(* Visualisation MANUAL_ST00_2
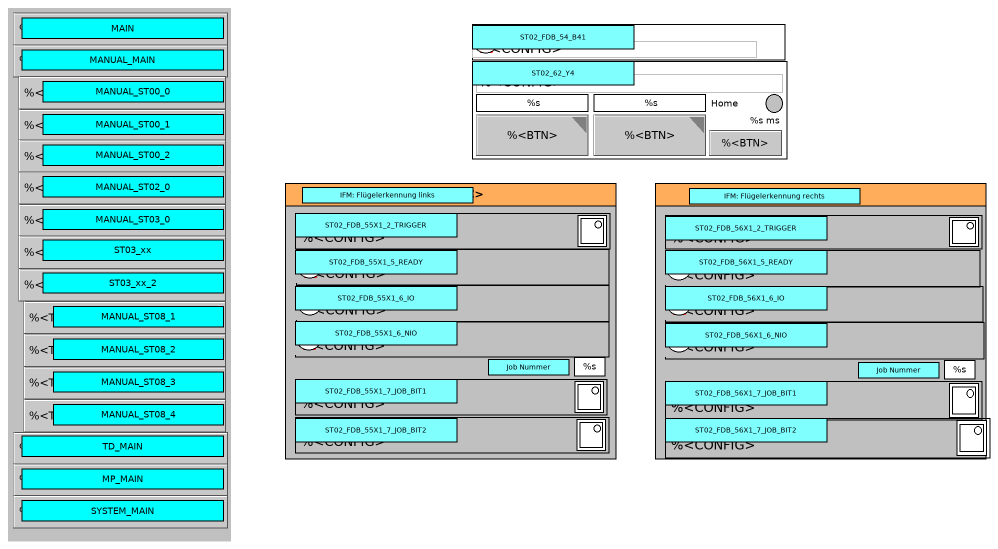
rectangle at (280,290)-(611,313): text "%<BASIC>"; shows 'IFM_Flügelerkennung_links'
rectangle at (650,290)-(981,313): text "%<BASIC>"; shows 'IFM_Flügelerkennung_rechts'
embedded screen at (3,115)-(226,648): M0000_Manual
embedded screen at (291,356)-(604,392): VDIGIN
embedded screen at (291,392)-(604,429): VDIGIN
embedded screen at (290,428)-(604,464): VDIGIN
embedded screen at (660,322)-(977,356): VDIGOUT_SMAL
embedded screen at (660,357)-(975,394): VDIGIN
embedded screen at (660,393)-(978,429): VDIGIN
embedded screen at (660,429)-(979,466): VDIGIN
embedded screen at (467,131)-(780,167): VDIGIN
embedded screen at (467,168)-(782,266): ZLIB_VALVE_1_SENSORS
embedded screen at (290,320)-(605,356): VDIGOUT_SMAL
embedded screen at (290,486)-(602,522): VDIGOUT_SMAL
embedded screen at (290,524)-(604,560): VDIGOUT_SMAL
embedded screen at (660,488)-(977,527): VDIGOUT_SMAL
embedded screen at (660,525)-(985,565): VDIGOUT_SMAL
rectangle at (297,294)-(468,310): text "IFM: Flügelerkennung links"; invisible if TRUE
rectangle at (684,295)-(855,311): text "IFM: Flügelerkennung rechts"; invisible if TRUE
rectangle at (481,464)-(562,483): text "%<BASIC>"; shows 'Job Nummer'
rectangle at (569,464)-(600,483): text "%s"; shows TD.IFM_CamProgNo; editable 0..3
rectangle at (483,466)-(564,482): text "Job Nummer"; invisible if TRUE
rectangle at (851,467)-(932,486): text "%<BASIC>"; shows 'Job Nummer'
rectangle at (939,467)-(970,486): text "%s"; shows TD.IFM_CamProgNo; editable 0..3
rectangle at (853,469)-(934,485): text "Job Nummer"; invisible if TRUE
rectangle at (290,486)-(452,510): text "ST02_FDB_55X1_7_JOB_BIT1"; invisible if TRUE
rectangle at (290,525)-(452,549): text "ST02_FDB_55X1_7_JOB_BIT2"; invisible if TRUE
rectangle at (290,428)-(452,452): text "ST02_FDB_55X1_6_NIO"; invisible if TRUE
rectangle at (290,393)-(452,417): text "ST02_FDB_55X1_6_IO"; invisible if TRUE
rectangle at (290,357)-(452,381): text "ST02_FDB_55X1_5_READY"; invisible if TRUE
rectangle at (290,320)-(452,344): text "ST02_FDB_55X1_2_TRIGGER"; invisible if TRUE
rectangle at (660,488)-(822,512): text "ST02_FDB_56X1_7_JOB_BIT1"; invisible if TRUE
rectangle at (660,525)-(822,549): text "ST02_FDB_56X1_7_JOB_BIT2"; invisible if TRUE
rectangle at (660,430)-(822,454): text "ST02_FDB_56X1_6_NIO"; invisible if TRUE
rectangle at (660,393)-(822,417): text "ST02_FDB_56X1_6_IO"; invisible if TRUE
rectangle at (660,357)-(822,381): text "ST02_FDB_56X1_5_READY"; invisible if TRUE
rectangle at (660,323)-(822,347): text "ST02_FDB_56X1_2_TRIGGER"; invisible if TRUE
rectangle at (467,132)-(629,156): text "ST02_FDB_54_B41"; invisible if TRUE
rectangle at (467,168)-(629,192): text "ST02_62_Y4"; invisible if TRUE
2 more shapes without text or variables
*)

(* Visualisation MANUAL_ST02_0
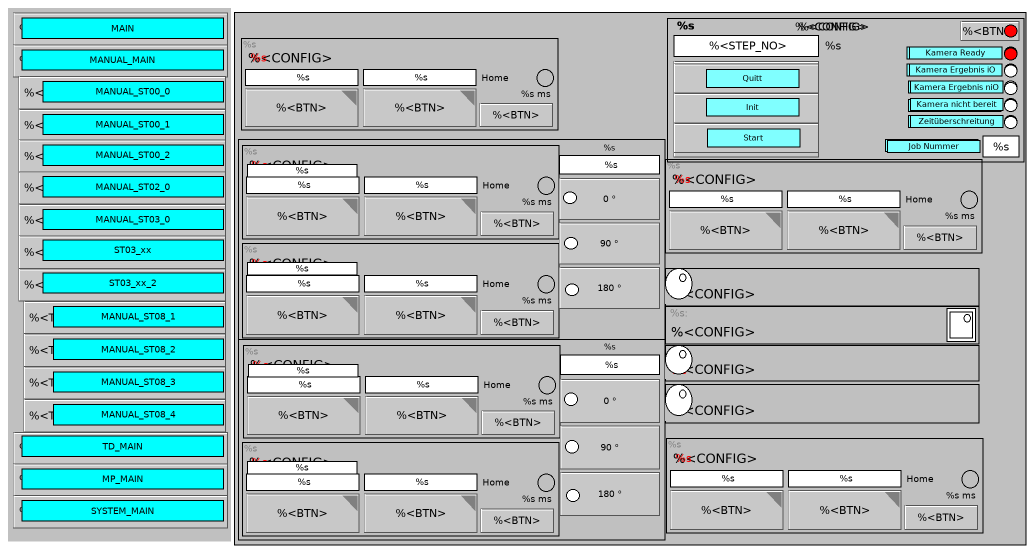
embedded screen at (3,115)-(226,648): M0000_Manual
rectangle at (233,246)-(660,447): alarm colour if ST02_62_Y6.SensorWorkIn[1].SensorSignal
rectangle at (233,446)-(660,647): alarm colour if ST02_62_Y6.SensorInitIn[1].SensorSignal
embedded screen at (660,413)-(974,451): VDIGOUT_SMAL
embedded screen at (236,145)-(553,237): ZLIB_VALVE_1_SENSORS
embedded screen at (660,452)-(974,488): VDIGIN
embedded screen at (237,350)-(554,445): ZLIB_VALVE_1_SENSORS
embedded screen at (237,252)-(554,346): ZLIB_VALVE_1_SENSORS
embedded screen at (237,549)-(554,643): ZLIB_VALVE_1_SENSORS
embedded screen at (238,452)-(555,545): ZLIB_VALVE_1_SENSORS
embedded screen at (552,249)-(657,422): ZLIB_Schwenkarm
embedded screen at (553,448)-(657,629): ZLIB_Schwenkarm
rectangle at (242,568)-(352,581): text "%s"; shows 'ST02_DT_61_B51'; alarm colour if ST02_DT_61_B51.ValveSensor
rectangle at (243,471)-(353,484): text "%s"; shows 'ST02_DT_61_B51'; alarm colour if ST02_DT_61_B51.ValveSensor
rectangle at (242,369)-(352,382): text "%s"; shows 'ST02_DT_61_B21'; alarm colour if ST02_DT_61_B21.ValveSensor
rectangle at (242,271)-(352,284): text "%s"; shows 'ST02_DT_61_B21'; alarm colour if ST02_DT_61_B21.ValveSensor
embedded screen at (660,375)-(974,413): VDIGIN
embedded screen at (660,491)-(974,530): VDIGIN
embedded screen at (661,545)-(978,640): ZLIB_VALVE_1_SENSORS
embedded screen at (660,266)-(977,360): ZLIB_VALVE_1_SENSORS
embedded screen at (662,125)-(1019,269): ZLIB_SENSOPART; invisible if MP.ST02.SensopartEthernet
embedded screen at (662,125)-(1019,269): ZLIB_SENSOPART_4; invisible if NOT MP.ST02.SensopartEthernet
1 more shapes without text or variables
*)

(* Visualisation MANUAL_ST03_0
embedded screen at (3,115)-(226,656): M0000_Manual
embedded screen at (234,123)-(549,159): VDIGIN
embedded screen at (233,161)-(844,458): ZLIB_EPSON_ROBOT
button at (244,538)-(555,574): text "%<BTN>"; shows 'Schwenkeinheit Ein'; taps ST03_ManRobotSwivelUnit.ToggleBtnOn; dynamic style Color.lightgrey, ModeSelect.Mode<>MODE_MANUAL OR NOT Robot01.RemInRunning
button at (244,462)-(555,498): text "%<BTN>"; shows 'Schwenkeinheit Aus'; taps ST03_ManRobotSwivelUnit.ToggleBtnOff; dynamic style Color.lightgrey, ModeSelect.Mode<>MODE_MANUAL OR NOT Robot01.RemInRunning
embedded screen at (244,499)-(559,536): VDIGIN
embedded screen at (244,575)-(559,612): VDIGIN
embedded screen at (244,615)-(559,652): VDIGIN; invisible if TRUE
rectangle at (244,538)-(351,557): text "Schwenkeinheit Ein"; invisible if TRUE
rectangle at (244,462)-(351,481): text "Schwenkeinheit Aus"; invisible if TRUE
rectangle at (235,124)-(407,145): text "ST03_125_F1"; invisible if TRUE
rectangle at (244,499)-(416,520): text "ST03_400_B12_6"; invisible if TRUE
rectangle at (244,575)-(416,596): text "ST03_400_B12_7"; invisible if TRUE
rectangle at (244,615)-(416,636): text "St03_120_A1_A14"; invisible if TRUE
rectangle at (0,0)-(111,51): text "%<BASIC>"; shows 'Lageerkennung'
rounded rectangle at (14,18)-(95,39): text "ERROR"
rounded rectangle at (14,18)-(95,39): text "Pos 35"; invisible if ST03_Init_AbholPos.RoboPos31 AND ST03_Init_AbholPos.RoboPos35
rounded rectangle at (14,18)-(95,39): text "Pos 31"; invisible if ST03_Init_AbholPos.RoboPos35; alarm colour if ST03_Init_AbholPos.RoboPos31
*)

(* Visualisation MANUAL_ST03_1
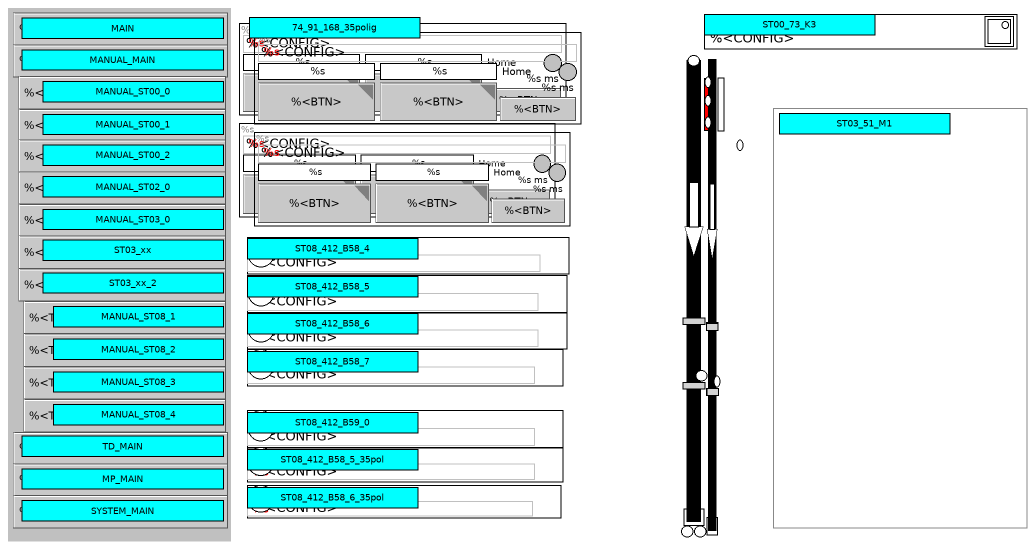
embedded screen at (3,115)-(226,648): M0000_Manual
embedded screen at (234,130)-(561,222): ZLIB_VALVE_1_SENSORS; invisible if MP.ST03.SGM_3621
embedded screen at (234,230)-(550,324): ZLIB_VALVE_1_SENSORS; invisible if MP.ST03.SGM_3621
embedded screen at (242,456)-(558,493): VDIGIN
embedded screen at (242,517)-(558,555): VDIGIN
embedded screen at (242,382)-(562,420): VDIGIN; invisible if gTypeCode = 4992
embedded screen at (242,419)-(562,456): VDIGIN; invisible if gTypeCode = 4992
embedded screen at (242,344)-(564,381): VDIGIN
embedded screen at (242,554)-(558,589): VDIGIN; invisible if gTypeCode <> 4992
embedded screen at (242,592)-(556,625): VDIGIN; invisible if gTypeCode <>4992
embedded screen at (670,162)-(711,644): ZUFUEHRUNG_35POL; invisible if gTypeCode <>4992
embedded screen at (697,166)-(738,642): ZUFUEHRUNG_74_91_168POL; invisible if gTypeCode<>360 AND gTypeCode <>379 AND gTypeCode <>489
other_LINEWIDTH at (768,215)-(1022,635): invisible if MP.ST03.SGM_3621
embedded screen at (249,139)-(576,231): ZLIB_VALVE_1_SENSORS; invisible if NOT MP.ST03.SGM_3621
embedded screen at (249,239)-(565,333): ZLIB_VALVE_1_SENSORS; invisible if NOT MP.ST03.SGM_3621
rectangle at (244,124)-(415,145): text "74_91_168_35polig"; invisible if TRUE
rectangle at (774,220)-(945,241): text "ST03_51_M1"; invisible if TRUE
rectangle at (242,345)-(413,366): text "ST08_412_B58_4"; invisible if TRUE
rectangle at (242,383)-(413,404): text "ST08_412_B58_5"; invisible if TRUE
rectangle at (242,420)-(413,441): text "ST08_412_B58_6"; invisible if TRUE
rectangle at (242,458)-(413,479): text "ST08_412_B58_7"; invisible if TRUE
rectangle at (242,519)-(413,540): text "ST08_412_B59_0"; invisible if TRUE
rectangle at (242,556)-(413,577): text "ST08_412_B58_5_35pol"; invisible if TRUE
rectangle at (242,594)-(413,615): text "ST08_412_B58_6_35pol"; invisible if TRUE
embedded screen at (699,121)-(1012,156): VDIGOUT_SMAL
rectangle at (699,121)-(870,142): text "ST00_73_K3"; invisible if TRUE
*)

(* Visualisation MANUAL_ST03_10
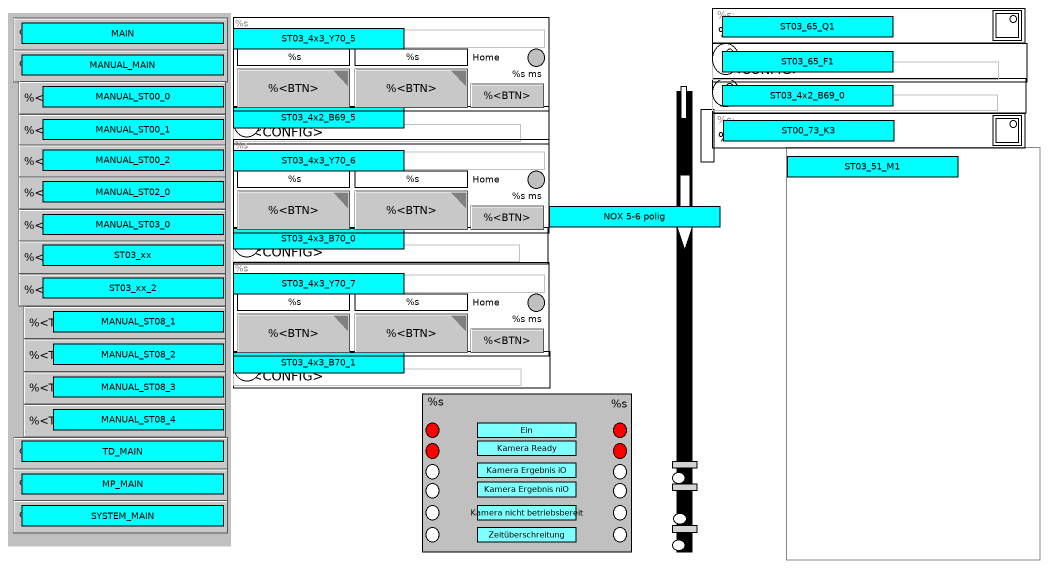
embedded screen at (3,115)-(226,648): M0000_Manual
embedded screen at (342,188)-(709,654): ZUFUEHRUNG_NOX_5_6POL; invisible if gTypeCode<>5632 AND gTypeCode<>5633
embedded screen at (228,453)-(545,490): VDIGIN
embedded screen at (707,180)-(1021,215): VDIGIN
embedded screen at (228,208)-(544,246): VDIGIN
embedded screen at (228,329)-(543,366): VDIGIN
rectangle at (544,308)-(715,329): text "NOX 5-6 polig"; invisible if TRUE
rectangle at (717,187)-(888,208): text "ST03_4x2_B69_0"; invisible if TRUE
rectangle at (228,209)-(399,230): text "ST03_4x2_B69_5"; invisible if TRUE
rectangle at (228,454)-(399,475): text "ST03_4x3_B70_1"; invisible if TRUE
rectangle at (228,330)-(399,351): text "ST03_4x3_B70_0"; invisible if TRUE
rectangle at (782,258)-(953,279): text "ST03_51_M1"; invisible if TRUE
embedded screen at (228,119)-(544,213): ZLIB_VALVE_1_SENSORS
rectangle at (228,130)-(399,151): text "ST03_4x3_Y70_5"; invisible if TRUE
embedded screen at (228,241)-(544,335): ZLIB_VALVE_1_SENSORS
rectangle at (228,252)-(399,273): text "ST03_4x3_Y70_6"; invisible if TRUE
embedded screen at (228,364)-(544,458): ZLIB_VALVE_1_SENSORS
rectangle at (228,375)-(399,396): text "ST03_4x3_Y70_7"; invisible if TRUE
embedded screen at (707,110)-(1020,145): VDIGOUT_SMAL
rectangle at (717,118)-(888,139): text "ST03_65_Q1"; invisible if TRUE
embedded screen at (707,145)-(1022,184): VDIGIN
rectangle at (717,153)-(888,174): text "ST03_65_F1"; invisible if TRUE
embedded screen at (707,215)-(1020,250): VDIGOUT_SMAL
rectangle at (718,222)-(889,243): text "ST00_73_K3"; invisible if TRUE
1 more shapes without text or variables
*)

(* Visualisation MANUAL_ST03_10_2
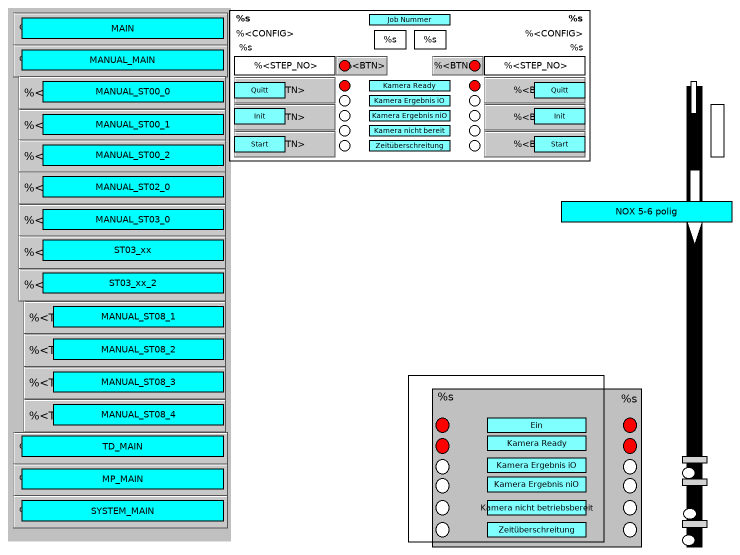
embedded screen at (3,115)-(226,648): M0000_Manual
embedded screen at (352,188)-(719,654): ZUFUEHRUNG_NOX_5_6POL; invisible if gTypeCode<>5632 AND gTypeCode<>5633
rectangle at (556,308)-(727,329): text "NOX 5-6 polig"; invisible if TRUE
embedded screen at (224,117)-(585,268): ZLIB_SENSOPART_4_2
1 more shapes without text or variables
*)

(* Visualisation MANUAL_ST03_11
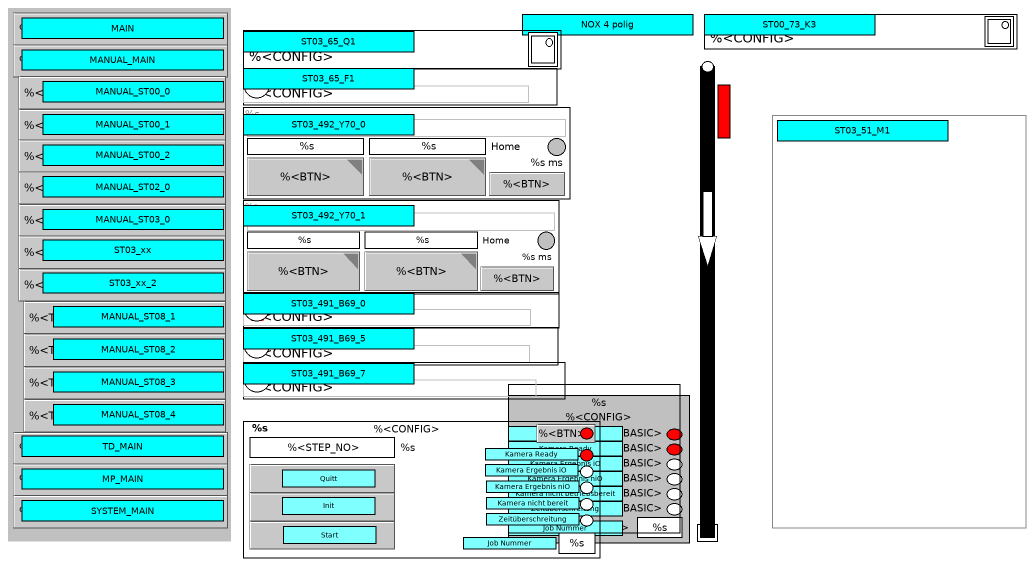
embedded screen at (3,115)-(226,648): M0000_Manual
embedded screen at (238,214)-(565,306): ZLIB_VALVE_1_SENSORS
embedded screen at (238,307)-(554,401): ZLIB_VALVE_1_SENSORS
embedded screen at (238,399)-(554,435): VDIGIN
embedded screen at (238,434)-(553,472): VDIGIN
embedded screen at (503,168)-(725,650): ZUFUEHRUNG_NOX_4POL; invisible if gTypeCode<>5631
rectangle at (517,121)-(688,142): text "NOX 4 polig"; invisible if TRUE
rectangle at (238,312)-(409,333): text "ST03_492_Y70_1"; invisible if TRUE
rectangle at (238,221)-(409,242): text "ST03_492_Y70_0"; invisible if TRUE
rectangle at (238,400)-(409,421): text "ST03_491_B69_0"; invisible if TRUE
rectangle at (238,435)-(409,456): text "ST03_491_B69_5"; invisible if TRUE
rectangle at (772,227)-(943,248): text "ST03_51_M1"; invisible if TRUE
embedded screen at (238,137)-(556,176): VDIGOUT_SMAL
rectangle at (238,138)-(409,159): text "ST03_65_Q1"; invisible if TRUE
embedded screen at (238,175)-(552,212): VDIGIN
rectangle at (238,175)-(409,196): text "ST03_65_F1"; invisible if TRUE
embedded screen at (699,121)-(1012,156): VDIGOUT_SMAL
rectangle at (699,121)-(870,142): text "ST00_73_K3"; invisible if TRUE
embedded screen at (238,528)-(595,665): ZLIB_SENSOPART_4; invisible if TRUE
embedded screen at (238,469)-(560,506): VDIGIN
rectangle at (238,470)-(409,491): text "ST03_491_B69_7"; invisible if TRUE
2 more shapes without text or variables
*)

(* Visualisation MANUAL_ST03_12
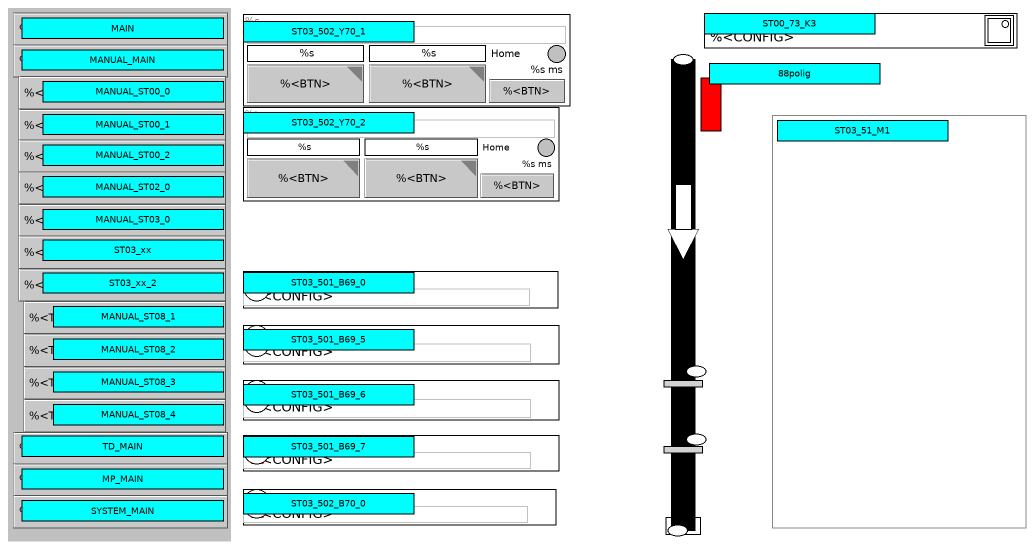
embedded screen at (3,115)-(226,648): M0000_Manual
embedded screen at (238,121)-(565,213): ZLIB_VALVE_1_SENSORS
embedded screen at (238,214)-(554,308): ZLIB_VALVE_1_SENSORS
embedded screen at (238,542)-(554,578): VDIGIN
embedded screen at (238,596)-(551,632): VDIGIN
embedded screen at (646,161)-(716,643): ZUFUEHRUNG_88POL; invisible if gTypeCode<>5731
rectangle at (704,170)-(875,191): text "88polig"; invisible if TRUE
rectangle at (238,219)-(409,240): text "ST03_502_Y70_2"; invisible if TRUE
rectangle at (238,128)-(409,149): text "ST03_502_Y70_1"; invisible if TRUE
rectangle at (238,543)-(409,564): text "ST03_501_B69_7"; invisible if TRUE
rectangle at (238,600)-(409,621): text "ST03_502_B70_0"; invisible if TRUE
rectangle at (772,227)-(943,248): text "ST03_51_M1"; invisible if TRUE
embedded screen at (238,487)-(554,527): VDIGIN
embedded screen at (238,378)-(553,415): VDIGIN
embedded screen at (238,432)-(554,471): VDIGIN
rectangle at (238,379)-(409,400): text "ST03_501_B69_0"; invisible if TRUE
rectangle at (238,436)-(409,457): text "ST03_501_B69_5"; invisible if TRUE
rectangle at (238,491)-(409,512): text "ST03_501_B69_6"; invisible if TRUE
embedded screen at (699,120)-(1012,155): VDIGOUT_SMAL
rectangle at (699,120)-(870,141): text "ST00_73_K3"; invisible if TRUE
1 more shapes without text or variables
*)

(* Visualisation MANUAL_ST03_13
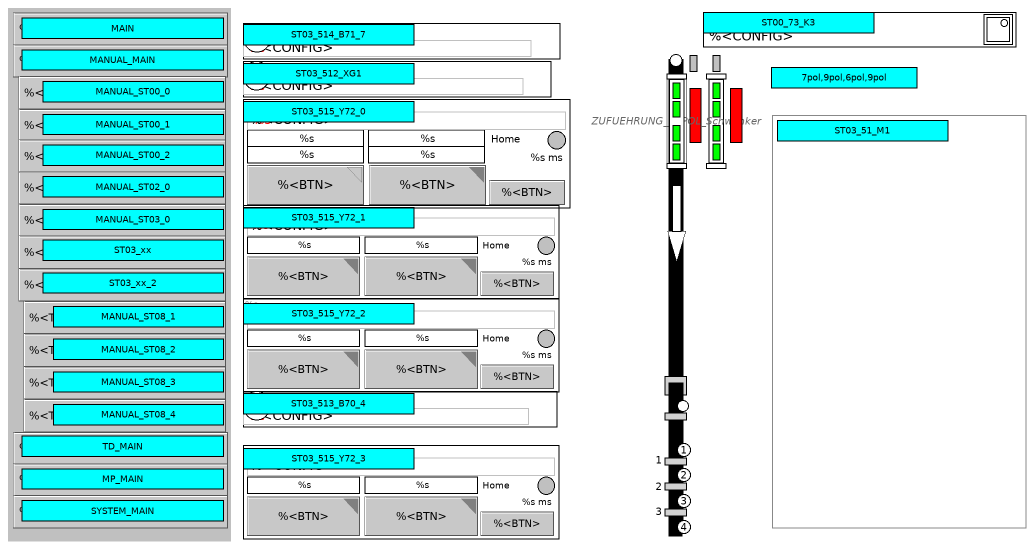
embedded screen at (3,115)-(226,648): M0000_Manual
embedded screen at (238,312)-(554,406): ZLIB_VALVE_1_SENSORS
embedded screen at (238,130)-(555,166): VDIGIN
embedded screen at (646,161)-(737,643): ZUFUEHRUNG_7POL; invisible if gTypeCode<>575  AND gTypeCode<>5753  AND gTypeCode<>5754  AND gTypeCode<>5755
rectangle at (766,174)-(912,195): text "7pol,9pol,6pol,9pol"; invisible if TRUE
rectangle at (238,314)-(409,335): text "ST03_515_Y72_1"; invisible if TRUE
rectangle at (238,131)-(409,152): text "ST03_514_B71_7"; invisible if TRUE
rectangle at (772,227)-(943,248): text "ST03_51_M1"; invisible if TRUE
embedded screen at (238,168)-(546,204): VDIGIN
rectangle at (238,170)-(409,191): text "ST03_512_XG1"; invisible if TRUE
embedded screen at (238,405)-(554,499): ZLIB_VALVE_1_SENSORS
embedded screen at (238,498)-(552,534): VDIGIN
rectangle at (238,410)-(409,431): text "ST03_515_Y72_2"; invisible if TRUE
rectangle at (238,500)-(409,521): text "ST03_513_B70_4"; invisible if TRUE
embedded screen at (238,552)-(554,646): ZLIB_VALVE_1_SENSORS
rectangle at (238,555)-(409,576): text "ST03_515_Y72_3"; invisible if TRUE
embedded screen at (238,206)-(565,315): ZLIB_VALVE_2_SENSORS
rectangle at (238,208)-(409,229): text "ST03_515_Y72_0"; invisible if TRUE
embedded screen at (698,119)-(1011,154): VDIGOUT_SMAL
rectangle at (698,119)-(869,140): text "ST00_73_K3"; invisible if TRUE
1 more shapes without text or variables
*)

(* Visualisation MANUAL_ST03_13_2
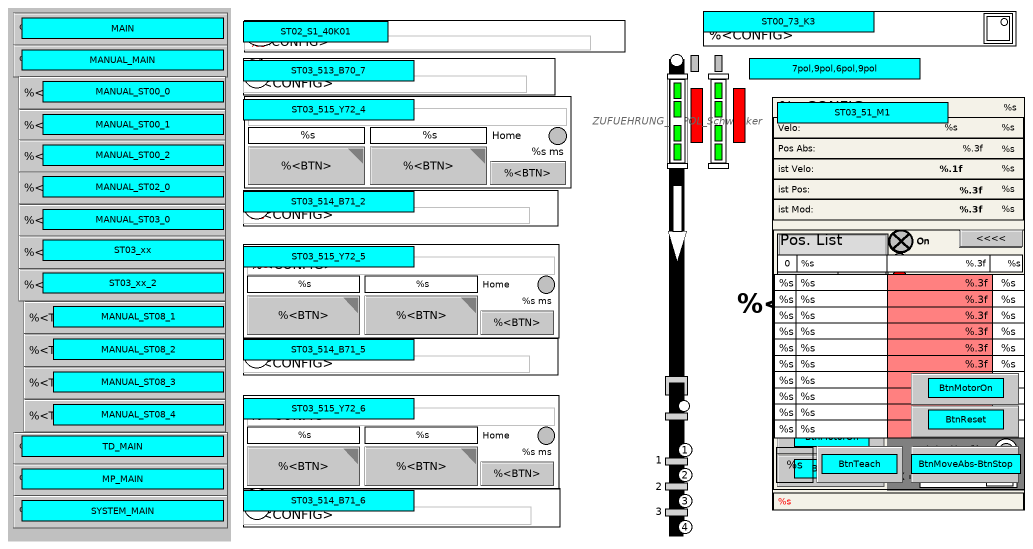
embedded screen at (3,115)-(226,648): M0000_Manual
embedded screen at (239,203)-(566,295): ZLIB_VALVE_1_SENSORS
embedded screen at (238,351)-(554,445): ZLIB_VALVE_1_SENSORS
embedded screen at (238,445)-(553,482): VDIGIN
embedded screen at (767,204)-(1021,617): ZLIB_7211_Achse
embedded screen at (646,161)-(740,643): ZUFUEHRUNG_7POL; invisible if gTypeCode<>575  AND gTypeCode<>5753  AND gTypeCode<>5754  AND gTypeCode<>5755
rectangle at (744,165)-(915,186): text "7pol,9pol,6pol,9pol"; invisible if TRUE
rectangle at (238,353)-(409,374): text "ST03_515_Y72_5"; invisible if TRUE
rectangle at (238,206)-(409,227): text "ST03_515_Y72_4"; invisible if TRUE
rectangle at (238,446)-(409,467): text "ST03_514_B71_5"; invisible if TRUE
rectangle at (772,209)-(943,230): text "ST03_51_M1"; invisible if TRUE
embedded screen at (238,165)-(550,202): VDIGIN
rectangle at (238,167)-(409,188): text "ST03_513_B70_7"; invisible if TRUE
embedded screen at (238,502)-(554,596): ZLIB_VALVE_1_SENSORS
embedded screen at (238,595)-(555,634): VDIGIN
rectangle at (238,505)-(409,526): text "ST03_515_Y72_6"; invisible if TRUE
rectangle at (238,597)-(409,618): text "ST03_514_B71_6"; invisible if TRUE
embedded screen at (238,297)-(553,333): VDIGIN
rectangle at (238,298)-(409,319): text "ST03_514_B71_2"; invisible if TRUE
embedded screen at (239,127)-(620,159): VDIGIN; invisible if gTypeCode<>4991 AND gTypeCode <>312
rectangle at (238,128)-(383,149): text "ST02_S1_40K01"; invisible if TRUE
embedded screen at (698,118)-(1011,153): VDIGOUT_SMAL
rectangle at (698,118)-(869,139): text "ST00_73_K3"; invisible if TRUE
*)

(* Visualisation MANUAL_ST03_14
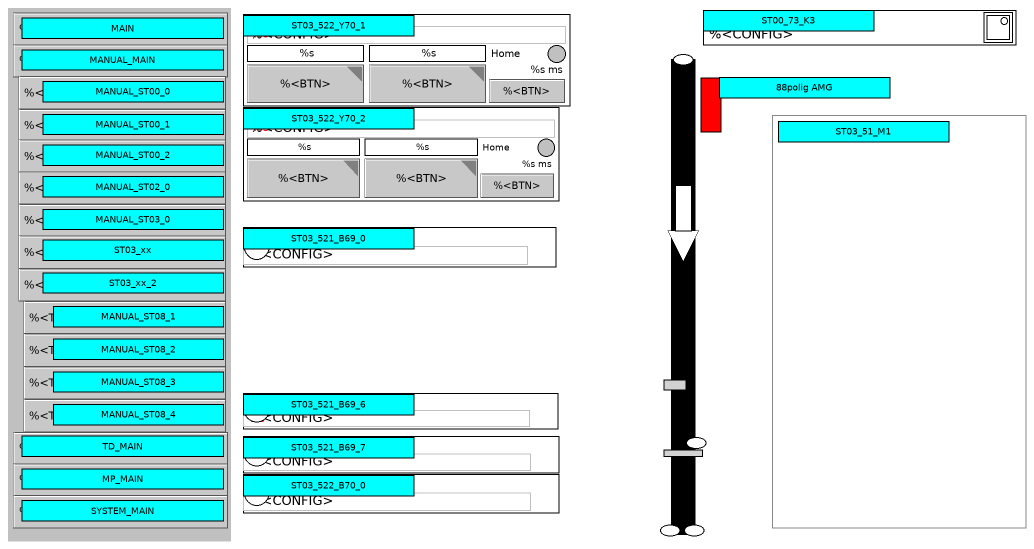
embedded screen at (3,115)-(226,648): M0000_Manual
embedded screen at (238,121)-(565,213): ZLIB_VALVE_1_SENSORS
embedded screen at (238,214)-(554,308): ZLIB_VALVE_1_SENSORS
embedded screen at (238,543)-(554,580): VDIGIN
embedded screen at (238,581)-(554,620): VDIGIN
embedded screen at (646,161)-(716,643): ZUFUEHRUNG_88POL_AMG; invisible if gTypeCode<>5732
rectangle at (714,184)-(885,205): text "88polig AMG"; invisible if TRUE
rectangle at (238,215)-(409,236): text "ST03_522_Y70_2"; invisible if TRUE
rectangle at (238,122)-(409,143): text "ST03_522_Y70_1"; invisible if TRUE
rectangle at (238,544)-(409,565): text "ST03_521_B69_7"; invisible if TRUE
rectangle at (238,582)-(409,603): text "ST03_522_B70_0"; invisible if TRUE
rectangle at (773,228)-(944,249): text "ST03_51_M1"; invisible if TRUE
embedded screen at (238,500)-(553,536): VDIGIN
embedded screen at (238,334)-(551,374): VDIGIN
rectangle at (238,335)-(409,356): text "ST03_521_B69_0"; invisible if TRUE
rectangle at (238,501)-(409,522): text "ST03_521_B69_6"; invisible if TRUE
embedded screen at (698,117)-(1011,152): VDIGOUT_SMAL
rectangle at (698,117)-(869,138): text "ST00_73_K3"; invisible if TRUE
1 more shapes without text or variables
*)

(* Visualisation MANUAL_ST03_15
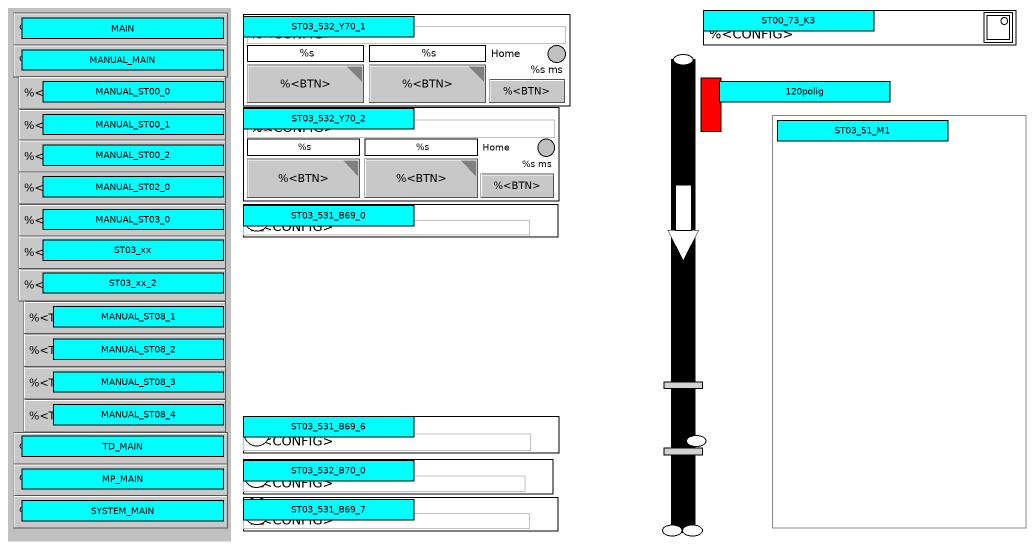
embedded screen at (3,115)-(226,648): M0000_Manual
embedded screen at (238,121)-(565,213): ZLIB_VALVE_1_SENSORS
embedded screen at (238,214)-(554,308): ZLIB_VALVE_1_SENSORS
embedded screen at (238,604)-(553,638): VDIGIN
embedded screen at (238,566)-(548,601): VDIGIN
embedded screen at (646,161)-(716,643): ZUFUEHRUNG_120POL; invisible if gTypeCode<>5771
rectangle at (714,188)-(885,209): text "120polig"; invisible if TRUE
rectangle at (238,215)-(409,236): text "ST03_532_Y70_2"; invisible if TRUE
rectangle at (238,123)-(409,144): text "ST03_532_Y70_1"; invisible if TRUE
rectangle at (238,606)-(409,627): text "ST03_531_B69_7"; invisible if TRUE
rectangle at (238,567)-(409,588): text "ST03_532_B70_0"; invisible if TRUE
rectangle at (772,227)-(943,248): text "ST03_51_M1"; invisible if TRUE
embedded screen at (238,523)-(554,560): VDIGIN
embedded screen at (238,311)-(553,344): VDIGIN
rectangle at (238,312)-(409,333): text "ST03_531_B69_0"; invisible if TRUE
rectangle at (238,523)-(409,544): text "ST03_531_B69_6"; invisible if TRUE
embedded screen at (698,117)-(1011,152): VDIGOUT_SMAL
rectangle at (698,117)-(869,138): text "ST00_73_K3"; invisible if TRUE
1 more shapes without text or variables
*)

(* Visualisation MANUAL_ST03_16
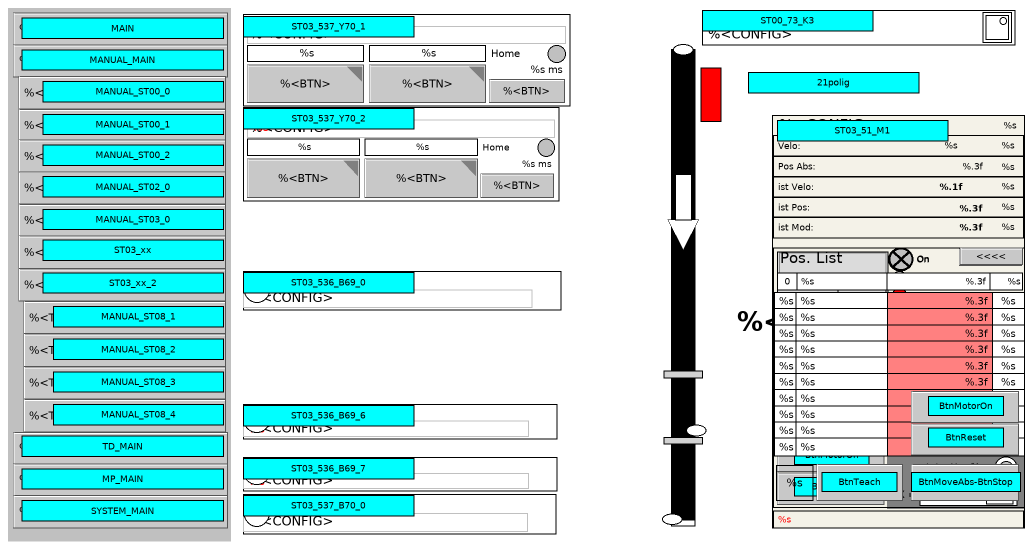
embedded screen at (3,115)-(226,648): M0000_Manual
embedded screen at (238,121)-(565,213): ZLIB_VALVE_1_SENSORS
embedded screen at (238,214)-(554,308): ZLIB_VALVE_1_SENSORS
embedded screen at (238,564)-(552,598): VDIGIN
embedded screen at (238,601)-(551,641): VDIGIN
embedded screen at (767,222)-(1021,635): ZLIB_7211_Achse
embedded screen at (646,151)-(716,633): ZUFUEHRUNG_21POL; invisible if gTypeCode<>5772
rectangle at (743,179)-(914,200): text "21polig"; invisible if TRUE
rectangle at (238,215)-(409,236): text "ST03_537_Y70_2"; invisible if TRUE
rectangle at (238,123)-(409,144): text "ST03_537_Y70_1"; invisible if TRUE
rectangle at (238,565)-(409,586): text "ST03_536_B69_7"; invisible if TRUE
rectangle at (238,602)-(409,623): text "ST03_537_B70_0"; invisible if TRUE
rectangle at (772,227)-(943,248): text "ST03_51_M1"; invisible if TRUE
embedded screen at (238,511)-(552,546): VDIGIN
embedded screen at (238,378)-(556,417): VDIGIN
rectangle at (238,379)-(409,400): text "ST03_536_B69_0"; invisible if TRUE
rectangle at (238,512)-(409,533): text "ST03_536_B69_6"; invisible if TRUE
embedded screen at (697,117)-(1010,152): VDIGOUT_SMAL
rectangle at (697,117)-(868,138): text "ST00_73_K3"; invisible if TRUE
*)

(* Visualisation MANUAL_ST03_17
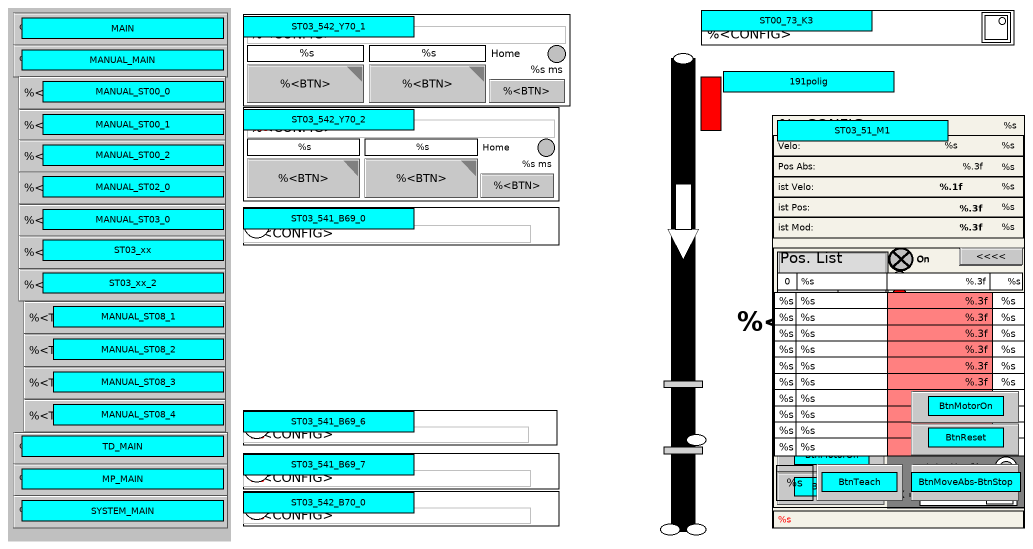
embedded screen at (3,115)-(226,648): M0000_Manual
embedded screen at (238,121)-(565,213): ZLIB_VALVE_1_SENSORS
embedded screen at (238,214)-(554,308): ZLIB_VALVE_1_SENSORS
embedded screen at (238,560)-(554,596): VDIGIN
embedded screen at (238,598)-(554,633): VDIGIN
embedded screen at (767,222)-(1021,635): ZLIB_7211_Achse
embedded screen at (646,160)-(716,642): ZUFUEHRUNG_191POL; invisible if gTypeCode<>580
rectangle at (718,178)-(889,199): text "191polig"; invisible if TRUE
rectangle at (238,216)-(409,237): text "ST03_542_Y70_2"; invisible if TRUE
rectangle at (238,123)-(409,144): text "ST03_542_Y70_1"; invisible if TRUE
rectangle at (238,561)-(409,582): text "ST03_541_B69_7"; invisible if TRUE
rectangle at (238,599)-(409,620): text "ST03_542_B70_0"; invisible if TRUE
rectangle at (772,227)-(943,248): text "ST03_51_M1"; invisible if TRUE
embedded screen at (238,517)-(552,552): VDIGIN
embedded screen at (238,314)-(554,352): VDIGIN
rectangle at (238,315)-(409,336): text "ST03_541_B69_0"; invisible if TRUE
rectangle at (238,518)-(409,539): text "ST03_541_B69_6"; invisible if TRUE
embedded screen at (696,117)-(1009,152): VDIGOUT_SMAL
rectangle at (696,117)-(867,138): text "ST00_73_K3"; invisible if TRUE
*)

(* Visualisation MANUAL_ST03_18
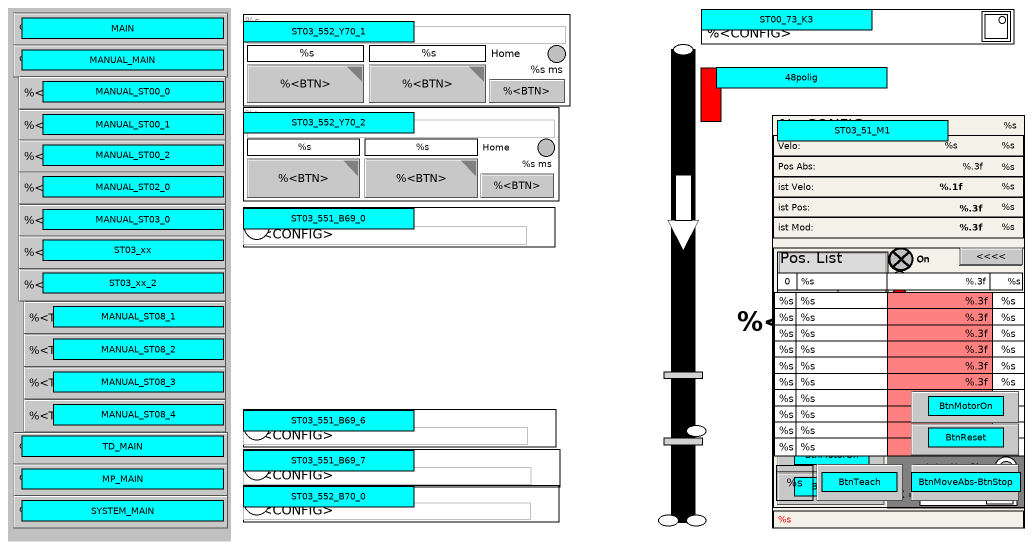
embedded screen at (3,115)-(226,648): M0000_Manual
embedded screen at (238,121)-(565,213): ZLIB_VALVE_1_SENSORS
embedded screen at (238,214)-(554,308): ZLIB_VALVE_1_SENSORS
embedded screen at (238,556)-(555,594): VDIGIN
embedded screen at (238,592)-(554,629): VDIGIN
embedded screen at (767,222)-(1021,635): ZLIB_7211_Achse
embedded screen at (646,151)-(716,633): ZUFUEHRUNG_48POL; invisible if gTypeCode<>5832
rectangle at (711,174)-(882,195): text "48polig"; invisible if TRUE
rectangle at (238,219)-(409,240): text "ST03_552_Y70_2"; invisible if TRUE
rectangle at (238,128)-(409,149): text "ST03_552_Y70_1"; invisible if TRUE
rectangle at (238,557)-(409,578): text "ST03_551_B69_7"; invisible if TRUE
rectangle at (238,593)-(409,614): text "ST03_552_B70_0"; invisible if TRUE
rectangle at (772,227)-(943,248): text "ST03_51_M1"; invisible if TRUE
embedded screen at (238,516)-(551,554): VDIGIN
embedded screen at (238,314)-(550,354): VDIGIN
rectangle at (238,315)-(409,336): text "ST03_551_B69_0"; invisible if TRUE
rectangle at (238,517)-(409,538): text "ST03_551_B69_6"; invisible if TRUE
embedded screen at (696,116)-(1009,151): VDIGOUT_SMAL
rectangle at (696,116)-(867,137): text "ST00_73_K3"; invisible if TRUE
*)

(* Visualisation MANUAL_ST03_19
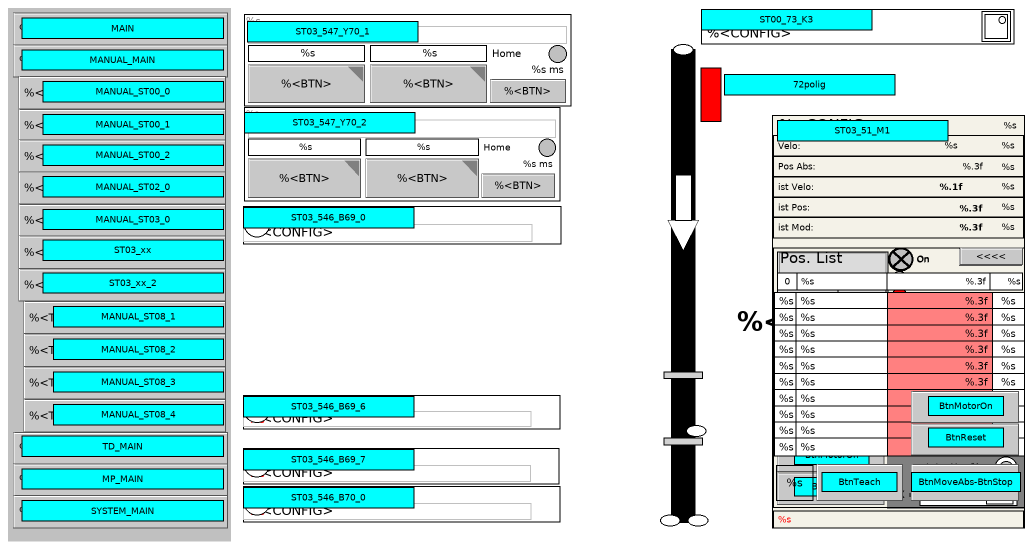
embedded screen at (3,115)-(226,648): M0000_Manual
embedded screen at (239,121)-(566,213): ZLIB_VALVE_1_SENSORS
embedded screen at (239,214)-(555,308): ZLIB_VALVE_1_SENSORS
embedded screen at (238,555)-(554,591): VDIGIN
embedded screen at (238,593)-(555,629): VDIGIN
embedded screen at (767,222)-(1021,635): ZLIB_7211_Achse
embedded screen at (646,151)-(716,633): ZUFUEHRUNG_72POL; invisible if gTypeCode<>5831
rectangle at (719,181)-(890,202): text "72polig"; invisible if TRUE
rectangle at (239,219)-(410,240): text "ST03_547_Y70_2"; invisible if TRUE
rectangle at (242,128)-(413,149): text "ST03_547_Y70_1"; invisible if TRUE
rectangle at (238,556)-(409,577): text "ST03_546_B69_7"; invisible if TRUE
rectangle at (238,594)-(409,615): text "ST03_546_B70_0"; invisible if TRUE
rectangle at (772,227)-(943,248): text "ST03_51_M1"; invisible if TRUE
embedded screen at (238,502)-(555,536): VDIGIN
embedded screen at (238,313)-(556,351): VDIGIN
rectangle at (238,314)-(409,335): text "ST03_546_B69_0"; invisible if TRUE
rectangle at (238,503)-(409,524): text "ST03_546_B69_6"; invisible if TRUE
embedded screen at (696,116)-(1009,151): VDIGOUT_SMAL
rectangle at (696,116)-(867,137): text "ST00_73_K3"; invisible if TRUE
*)

(* Visualisation MANUAL_ST03_2
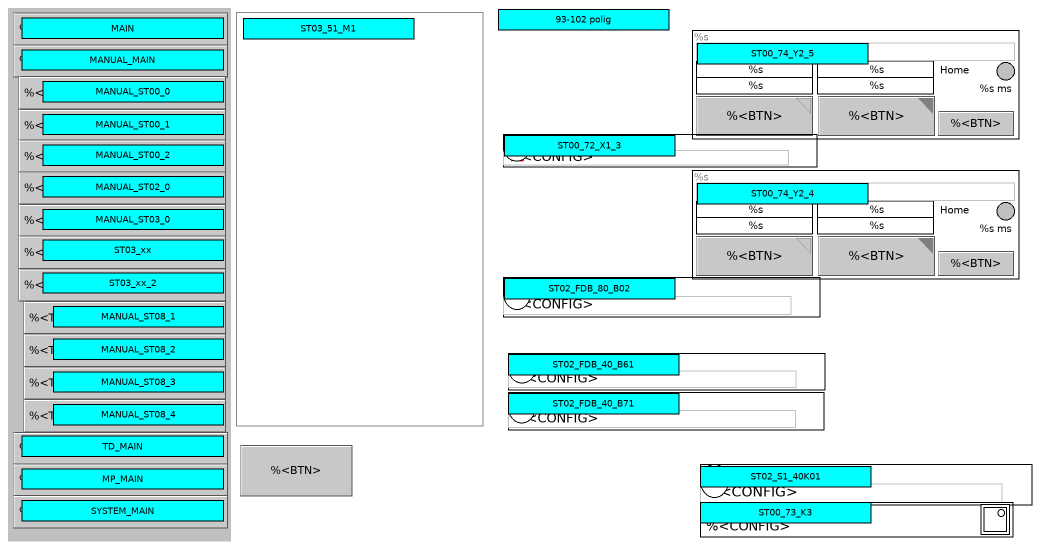
embedded screen at (3,115)-(226,648): M0000_Manual
embedded screen at (687,277)-(1014,386): ZLIB_VALVE_2_SENSORS
embedded screen at (687,137)-(1014,246): ZLIB_VALVE_2_SENSORS
other_LINEWIDTH at (231,119)-(478,533): invisible if MP.ST03.SGM_3621
embedded screen at (695,571)-(1027,612): VDIGIN
embedded screen at (498,241)-(812,274): VDIGIN
embedded screen at (498,384)-(815,424): VDIGIN
button at (235,552)-(347,603): text "%<BTN>"; shows 'TaktBand'; invisible if gTypeCode<>4991 AND gTypeCode <>312; taps ST03_Band.b_MoveRel
embedded screen at (503,460)-(820,497): VDIGIN
embedded screen at (503,499)-(819,537): VDIGIN
rectangle at (493,116)-(664,137): text "93-102 polig"; invisible if TRUE
rectangle at (238,125)-(409,146): text "ST03_51_M1"; invisible if TRUE
rectangle at (695,573)-(866,594): text "ST02_S1_40K01"; invisible if TRUE
rectangle at (503,461)-(674,482): text "ST02_FDB_40_B61"; invisible if TRUE
rectangle at (503,500)-(674,521): text "ST02_FDB_40_B71"; invisible if TRUE
rectangle at (499,385)-(670,406): text "ST02_FDB_80_B02"; invisible if TRUE
rectangle at (499,242)-(670,263): text "ST00_72_X1_3"; invisible if TRUE
rectangle at (692,150)-(863,171): text "ST00_74_Y2_5"; invisible if TRUE
rectangle at (692,290)-(863,311): text "ST00_74_Y2_4"; invisible if TRUE
embedded screen at (695,609)-(1008,644): VDIGOUT_SMAL
rectangle at (695,609)-(866,630): text "ST00_73_K3"; invisible if TRUE
*)

(* Visualisation MANUAL_ST03_20
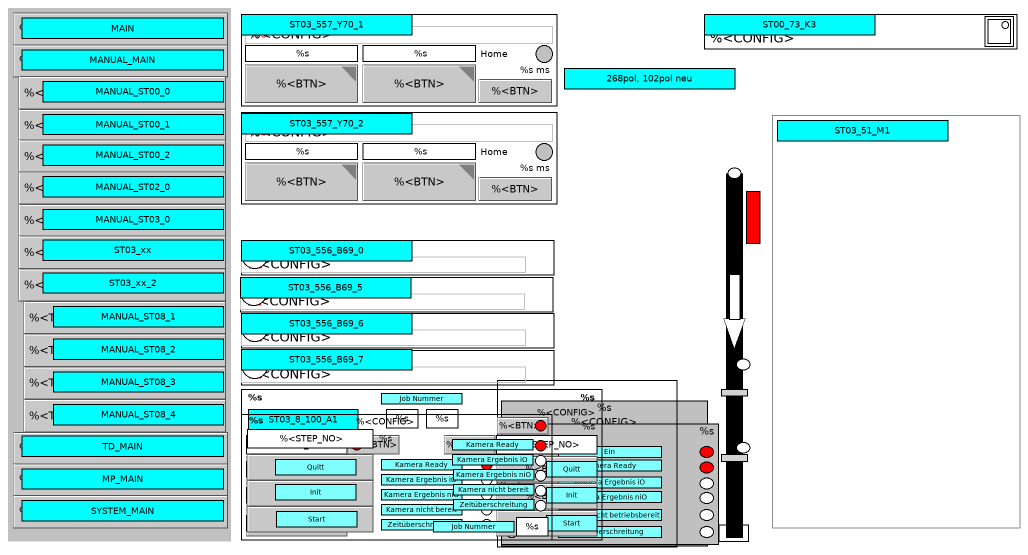
embedded screen at (3,115)-(226,648): M0000_Manual
embedded screen at (699,121)-(1012,156): VDIGOUT_SMAL
embedded screen at (236,121)-(552,213): ZLIB_VALVE_1_SENSORS
embedded screen at (236,219)-(552,311): ZLIB_VALVE_1_SENSORS
embedded screen at (496,176)-(755,653): ZUFUEHRUNG_268POL_102POL_NEU; invisible if AND gTypeCode<>4993
rectangle at (559,175)-(730,196): text "268pol, 102pol neu"; invisible if TRUE
rectangle at (236,220)-(407,241): text "ST03_557_Y70_2"; invisible if TRUE
rectangle at (236,121)-(407,142): text "ST03_557_Y70_1"; invisible if TRUE
rectangle at (699,121)-(870,142): text "ST00_73_K3"; invisible if TRUE
rectangle at (772,227)-(943,248): text "ST03_51_M1"; invisible if TRUE
embedded screen at (236,420)-(549,455): VDIGIN
embedded screen at (236,347)-(549,382): VDIGIN
rectangle at (236,347)-(407,368): text "ST03_556_B69_0"; invisible if TRUE
rectangle at (236,420)-(407,441): text "ST03_556_B69_6"; invisible if TRUE
embedded screen at (236,496)-(597,647): ZLIB_SENSOPART_4_2; invisible if gTypeCode<>4993
embedded screen at (235,384)-(548,419): VDIGIN
rectangle at (235,384)-(406,405): text "ST03_556_B69_5"; invisible if TRUE
rectangle at (243,516)-(353,537): text "ST03_8_100_A1"; invisible if TRUE
embedded screen at (236,457)-(549,492): VDIGIN
rectangle at (236,456)-(407,477): text "ST03_556_B69_7"; invisible if TRUE
embedded screen at (236,521)-(547,647): ZLIB_SENSOPART_4; invisible if gTypeCode<>5841
2 more shapes without text or variables
*)

(* Visualisation MANUAL_ST03_20_2
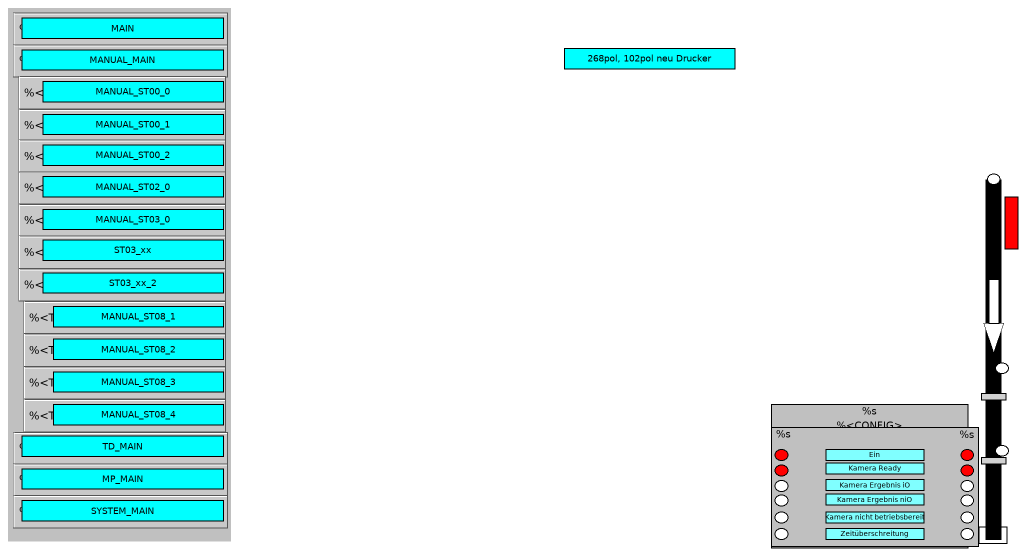
embedded screen at (766,183)-(1013,655): ZUFUEHRUNG_268POL_102POL_NEU
embedded screen at (3,115)-(226,648): M0000_Manual
rectangle at (559,155)-(730,176): text "268pol, 102pol neu Drucker"; invisible if TRUE
*)

(* Visualisation MANUAL_ST03_21
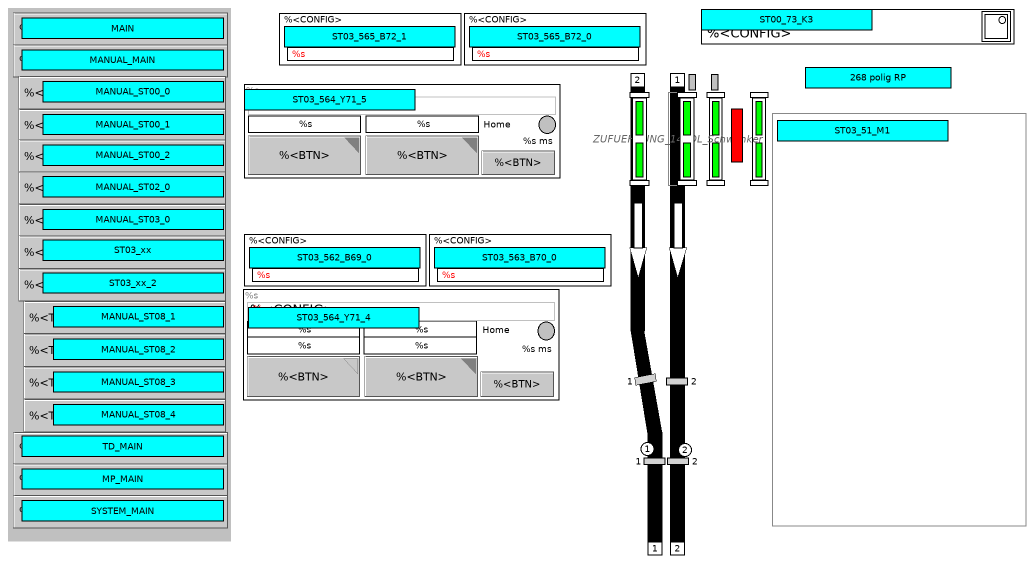
embedded screen at (3,115)-(226,648): M0000_Manual
embedded screen at (239,191)-(555,285): ZLIB_VALVE_1_SENSORS
embedded screen at (459,120)-(641,172): ZLIB_DIG_IN
embedded screen at (590,180)-(763,662): ZUFUEHRUNG_268POL_RP; invisible if gTypeCode<>5842
rectangle at (800,174)-(946,195): text "268 polig RP"; invisible if TRUE
rectangle at (239,196)-(410,217): text "ST03_564_Y71_5"; invisible if TRUE
rectangle at (464,133)-(635,154): text "ST03_565_B72_0"; invisible if TRUE
rectangle at (772,227)-(943,248): text "ST03_51_M1"; invisible if TRUE
embedded screen at (274,120)-(456,172): ZLIB_DIG_IN
rectangle at (279,133)-(450,154): text "ST03_565_B72_1"; invisible if TRUE
embedded screen at (239,341)-(421,393): ZLIB_DIG_IN
rectangle at (244,354)-(415,375): text "ST03_562_B69_0"; invisible if TRUE
embedded screen at (238,396)-(554,507): ZLIB_VALVE_2_SENSORS
rectangle at (243,414)-(414,435): text "ST03_564_Y71_4"; invisible if TRUE
embedded screen at (424,341)-(606,393): ZLIB_DIG_IN
rectangle at (429,354)-(600,375): text "ST03_563_B70_0"; invisible if TRUE
embedded screen at (696,116)-(1009,151): VDIGOUT_SMAL
rectangle at (696,116)-(867,137): text "ST00_73_K3"; invisible if TRUE
1 more shapes without text or variables
*)

(* Visualisation MANUAL_ST03_21_2
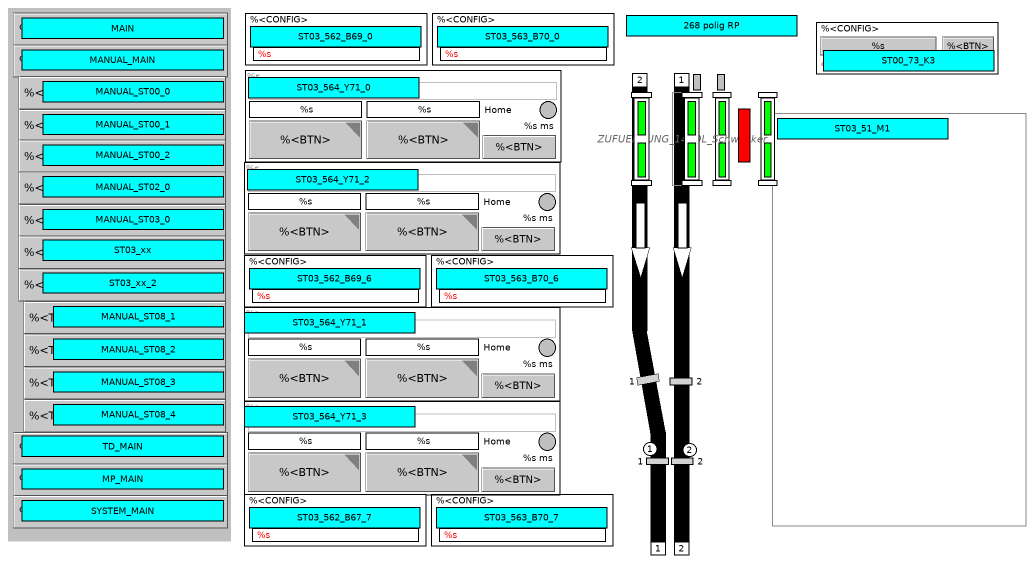
embedded screen at (3,115)-(226,648): M0000_Manual
embedded screen at (811,129)-(993,181): ZLIB_DIGOUT
embedded screen at (239,269)-(555,361): ZLIB_VALVE_1_SENSORS
embedded screen at (239,414)-(555,508): ZLIB_VALVE_1_SENSORS
embedded screen at (426,601)-(608,653): ZLIB_DIG_IN
embedded screen at (590,180)-(772,662): ZUFUEHRUNG_268POL_RP; invisible if gTypeCode<>5842
rectangle at (621,122)-(792,143): text "268 polig RP"; invisible if TRUE
rectangle at (239,419)-(410,440): text "ST03_564_Y71_1"; invisible if TRUE
rectangle at (242,276)-(413,297): text "ST03_564_Y71_2"; invisible if TRUE
rectangle at (431,614)-(602,635): text "ST03_563_B70_7"; invisible if TRUE
rectangle at (818,157)-(989,178): text "ST00_73_K3"; invisible if TRUE
rectangle at (772,225)-(943,246): text "ST03_51_M1"; invisible if TRUE
embedded screen at (426,362)-(608,414): ZLIB_DIG_IN
rectangle at (431,375)-(602,396): text "ST03_563_B70_6"; invisible if TRUE
embedded screen at (239,508)-(555,602): ZLIB_VALVE_1_SENSORS
embedded screen at (239,601)-(421,653): ZLIB_DIG_IN
rectangle at (239,513)-(410,534): text "ST03_564_Y71_3"; invisible if TRUE
rectangle at (244,614)-(415,635): text "ST03_562_B67_7"; invisible if TRUE
embedded screen at (239,362)-(421,414): ZLIB_DIG_IN
rectangle at (244,375)-(415,396): text "ST03_562_B69_6"; invisible if TRUE
embedded screen at (240,177)-(556,269): ZLIB_VALVE_1_SENSORS
rectangle at (243,184)-(414,205): text "ST03_564_Y71_0"; invisible if TRUE
embedded screen at (427,120)-(609,172): ZLIB_DIG_IN
rectangle at (432,133)-(603,154): text "ST03_563_B70_0"; invisible if TRUE
embedded screen at (240,120)-(422,172): ZLIB_DIG_IN
rectangle at (245,133)-(416,154): text "ST03_562_B69_0"; invisible if TRUE
1 more shapes without text or variables
*)

(* Visualisation MANUAL_ST03_22
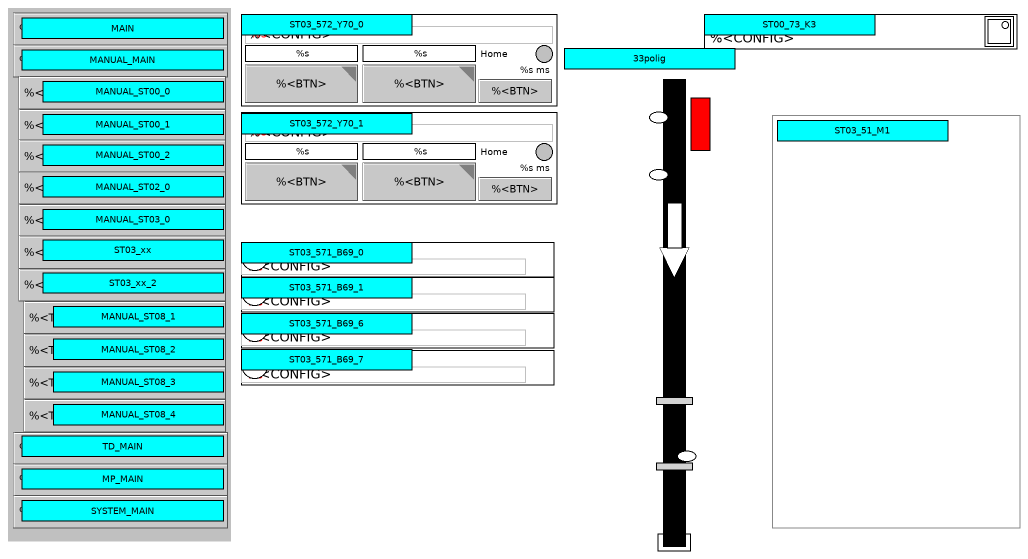
embedded screen at (3,115)-(226,648): M0000_Manual
embedded screen at (699,121)-(1012,156): VDIGOUT_SMAL
embedded screen at (236,121)-(552,213): ZLIB_VALVE_1_SENSORS
embedded screen at (236,219)-(552,311): ZLIB_VALVE_1_SENSORS
embedded screen at (236,457)-(549,492): VDIGIN
embedded screen at (639,181)-(705,658): ZUFUEHRUNG_33POL; invisible if gTypeCode<>598
rectangle at (559,155)-(730,176): text "33polig"; invisible if TRUE
rectangle at (236,220)-(407,241): text "ST03_572_Y70_1"; invisible if TRUE
rectangle at (236,121)-(407,142): text "ST03_572_Y70_0"; invisible if TRUE
rectangle at (236,456)-(407,477): text "ST03_571_B69_7"; invisible if TRUE
rectangle at (699,121)-(870,142): text "ST00_73_K3"; invisible if TRUE
rectangle at (772,227)-(943,248): text "ST03_51_M1"; invisible if TRUE
embedded screen at (236,420)-(549,455): VDIGIN
embedded screen at (236,384)-(549,419): VDIGIN
rectangle at (236,384)-(407,405): text "ST03_571_B69_1"; invisible if TRUE
rectangle at (236,420)-(407,441): text "ST03_571_B69_6"; invisible if TRUE
embedded screen at (236,349)-(549,384): VDIGIN
rectangle at (236,349)-(407,370): text "ST03_571_B69_0"; invisible if TRUE
1 more shapes without text or variables
*)

(* Visualisation MANUAL_ST03_23
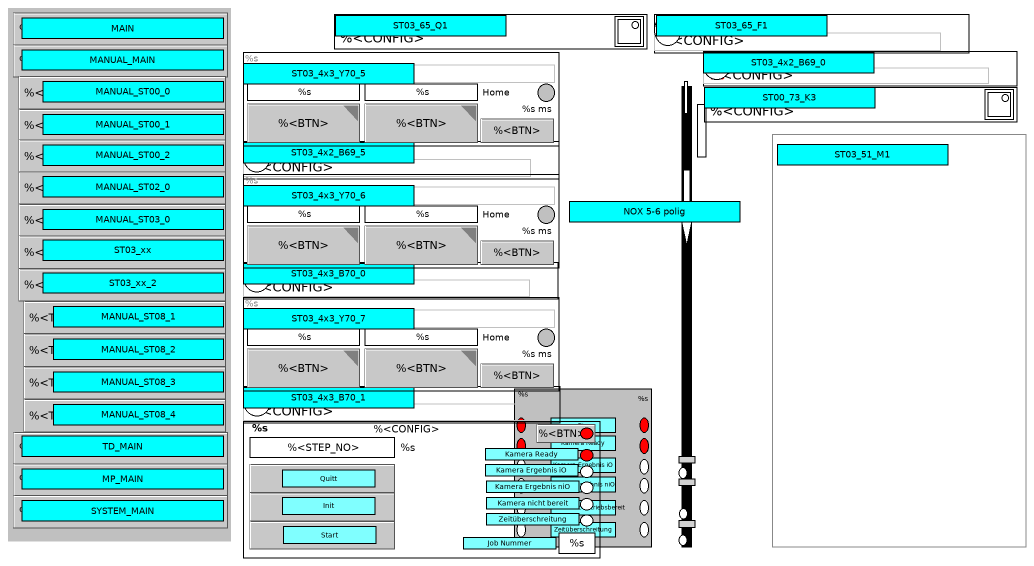
embedded screen at (3,115)-(226,648): M0000_Manual
embedded screen at (460,188)-(701,654): ZUFUEHRUNG_NOX_5_6POL; invisible if gTypeCode<>5632 AND gTypeCode<>5633
embedded screen at (238,493)-(555,530): VDIGIN
embedded screen at (698,158)-(1012,193): VDIGIN
embedded screen at (238,248)-(554,286): VDIGIN
embedded screen at (238,369)-(553,406): VDIGIN
rectangle at (564,308)-(735,329): text "NOX 5-6 polig"; invisible if TRUE
rectangle at (698,159)-(869,180): text "ST03_4x2_B69_0"; invisible if TRUE
rectangle at (238,249)-(409,270): text "ST03_4x2_B69_5"; invisible if TRUE
rectangle at (238,494)-(409,515): text "ST03_4x3_B70_1"; invisible if TRUE
rectangle at (238,370)-(409,391): text "ST03_4x3_B70_0"; invisible if TRUE
rectangle at (772,251)-(943,272): text "ST03_51_M1"; invisible if TRUE
embedded screen at (238,159)-(554,253): ZLIB_VALVE_1_SENSORS
rectangle at (238,170)-(409,191): text "ST03_4x3_Y70_5"; invisible if TRUE
embedded screen at (238,281)-(554,375): ZLIB_VALVE_1_SENSORS
rectangle at (238,292)-(409,313): text "ST03_4x3_Y70_6"; invisible if TRUE
embedded screen at (238,404)-(554,498): ZLIB_VALVE_1_SENSORS
rectangle at (238,415)-(409,436): text "ST03_4x3_Y70_7"; invisible if TRUE
embedded screen at (329,121)-(642,156): VDIGOUT_SMAL
rectangle at (330,122)-(501,143): text "ST03_65_Q1"; invisible if TRUE
embedded screen at (649,121)-(964,160): VDIGIN
rectangle at (651,122)-(822,143): text "ST03_65_F1"; invisible if TRUE
embedded screen at (699,194)-(1012,229): VDIGOUT_SMAL
rectangle at (699,194)-(870,215): text "ST00_73_K3"; invisible if TRUE
embedded screen at (238,528)-(595,665): ZLIB_SENSOPART_4
1 more shapes without text or variables
*)

(* Visualisation MANUAL_ST03_3
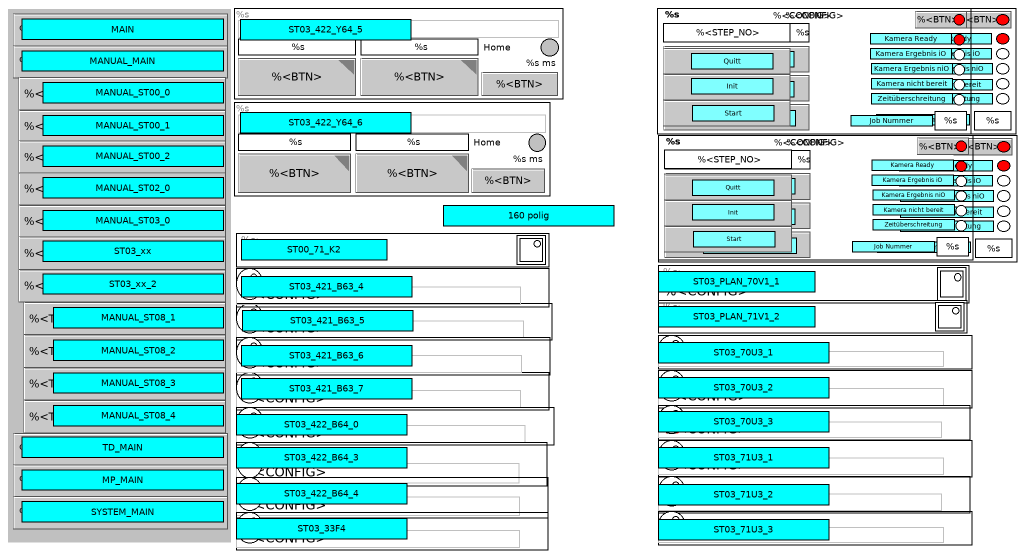
embedded screen at (3,115)-(226,648): M0000_MANUAL
embedded screen at (653,371)-(964,409): VDIGOUT_SMAL
embedded screen at (229,114)-(558,205): ZLIB_VALVE_1_SENSORS
embedded screen at (229,208)-(545,302): ZLIB_VALVE_1_SENSORS
embedded screen at (231,478)-(544,516): VDIGIN
embedded screen at (231,513)-(549,551): VDIGIN
embedded screen at (231,409)-(547,446): VDIGIN
embedded screen at (231,443)-(545,481): VDIGIN
embedded screen at (231,374)-(544,413): VDIGIN
embedded screen at (231,548)-(542,592): VDIGIN
embedded screen at (652,114)-(1011,240): ZLIB_SENSOPART
embedded screen at (653,241)-(1012,368): ZLIB_SENSOPART
embedded screen at (231,583)-(543,624): VDIGIN
embedded screen at (653,406)-(962,439): VDIGOUT_SMAL
embedded screen at (231,618)-(543,656): VDIGIN
embedded screen at (653,546)-(967,583): VDIGIN
embedded screen at (653,476)-(967,514): VDIGIN
embedded screen at (653,511)-(965,546): VDIGIN
embedded screen at (653,441)-(967,475): VDIGIN
embedded screen at (653,582)-(965,619): VDIGIN
embedded screen at (653,617)-(967,651): VDIGIN
embedded screen at (652,114)-(966,240): ZLIB_SENSOPART_4; invisible if NOT MP.ST02.SensopartEthernet
embedded screen at (653,241)-(968,366): ZLIB_SENSOPART_4; invisible if NOT MP.ST02.SensopartEthernet
rectangle at (438,311)-(609,332): text "160 polig"; invisible if TRUE
rectangle at (235,125)-(406,146): text "ST03_422_Y64_5"; invisible if TRUE
rectangle at (235,218)-(406,239): text "ST03_422_Y64_6"; invisible if TRUE
rectangle at (236,382)-(407,403): text "ST03_421_B63_4"; invisible if TRUE
rectangle at (231,520)-(402,541): text "ST03_422_B64_0"; invisible if TRUE
rectangle at (231,553)-(402,574): text "ST03_422_B64_3"; invisible if TRUE
rectangle at (237,416)-(408,437): text "ST03_421_B63_5"; invisible if TRUE
rectangle at (236,451)-(407,472): text "ST03_421_B63_6"; invisible if TRUE
rectangle at (231,589)-(402,610): text "ST03_422_B64_4"; invisible if TRUE
rectangle at (231,624)-(402,645): text "ST03_33F4"; invisible if TRUE
rectangle at (236,484)-(407,505): text "ST03_421_B63_7"; invisible if TRUE
rectangle at (653,448)-(824,469): text "ST03_70U3_1"; invisible if TRUE
rectangle at (653,483)-(824,504): text "ST03_70U3_2"; invisible if TRUE
rectangle at (653,517)-(824,538): text "ST03_70U3_3"; invisible if TRUE
rectangle at (653,553)-(824,574): text "ST03_71U3_1"; invisible if TRUE
rectangle at (653,590)-(824,611): text "ST03_71U3_2"; invisible if TRUE
rectangle at (653,625)-(824,646): text "ST03_71U3_3"; invisible if TRUE
rectangle at (653,377)-(810,398): text "ST03_PLAN_70V1_1"; invisible if TRUE
rectangle at (653,412)-(810,433): text "ST03_PLAN_71V1_2"; invisible if TRUE
embedded screen at (231,339)-(544,373): VDIGOUT_SMAL
rectangle at (236,345)-(382,366): text "ST00_71_K2"; invisible if TRUE
*)

(* Visualisation MANUAL_ST03_3_2
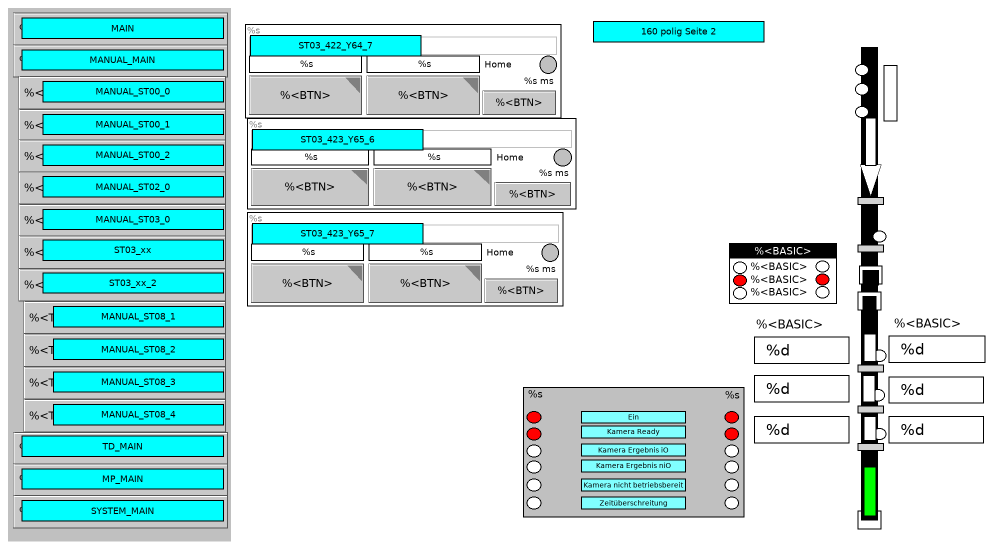
embedded screen at (3,115)-(226,648): M0000_MANUAL
embedded screen at (242,225)-(571,316): ZLIB_VALVE_1_SENSORS
embedded screen at (242,319)-(558,413): ZLIB_VALVE_1_SENSORS
embedded screen at (240,131)-(556,225): ZLIB_VALVE_1_SENSORS
rectangle at (588,128)-(759,149): text "160 polig Seite 2"; invisible if TRUE
embedded screen at (518,154)-(980,636): ZUFUEHRUNG_160POL; invisible if gTypeCode <>4992
rectangle at (245,142)-(416,163): text "ST03_422_Y64_7"; invisible if TRUE
rectangle at (247,236)-(418,257): text "ST03_423_Y65_6"; invisible if TRUE
rectangle at (247,330)-(418,351): text "ST03_423_Y65_7"; invisible if TRUE
*)

(* Visualisation MANUAL_ST03_4
